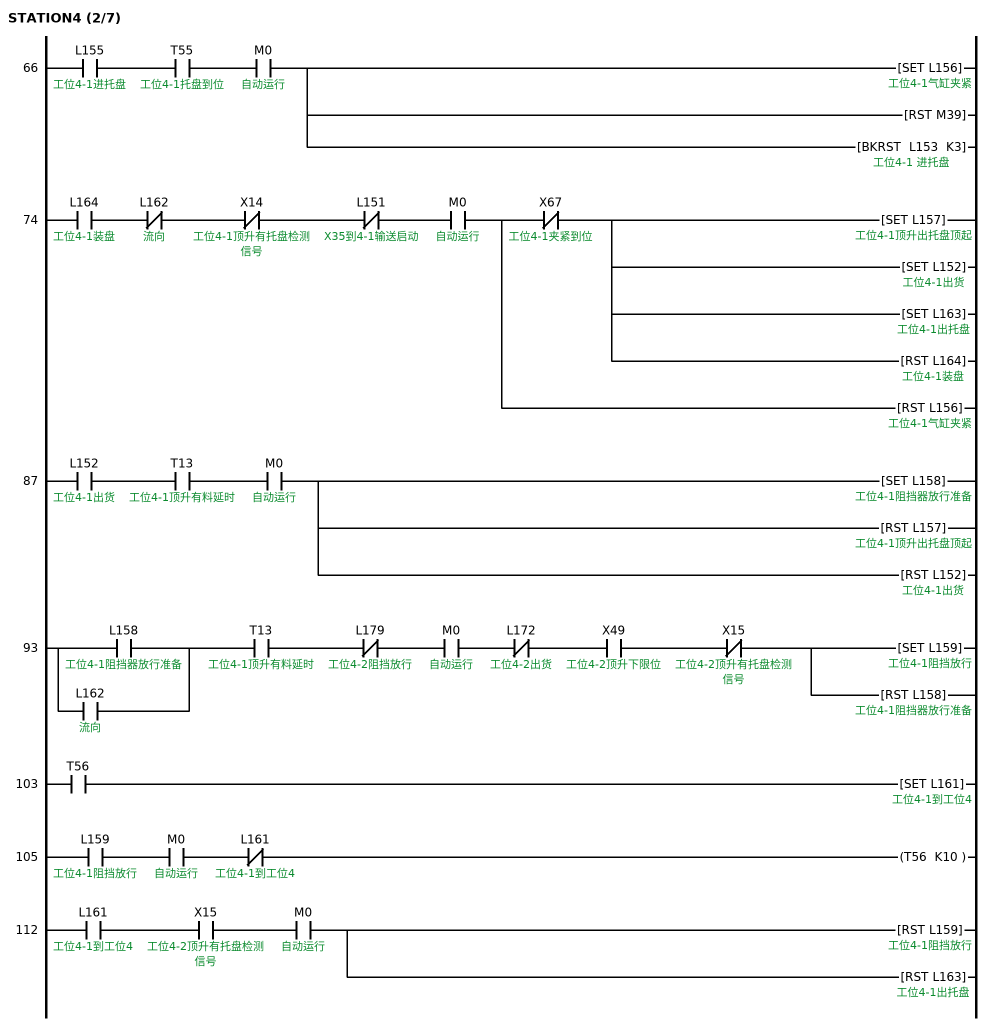
[picture p48: ladder of STATION4, rungs at steps 66 to 112]
66    LD      L155  ; 工位4-1进托盘
      AND     T55  ; 工位4-1托盘到位
      AND     M0  ; 自动运行
      SET     L156  ; 工位4-1气缸夹紧
      RST     M39
      BKRST   L153 K3
74    LD      L164  ; 工位4-1装盘
      ANI     L162  ; 流向
      ANI     X14  ; 工位4-1顶升有托盘检测信号
      ANI     L151  ; X35到4-1输送启动
      AND     M0  ; 自动运行
      MPS
      ANI     X67  ; 工位4-1夹紧到位
      SET     L157  ; 工位4-1顶升出托盘顶起
      SET     L152  ; 工位4-1出货
      SET     L163  ; 工位4-1出托盘
      RST     L164  ; 工位4-1装盘
      MPP
      RST     L156  ; 工位4-1气缸夹紧
87    LD      L152  ; 工位4-1出货
      AND     T13  ; 工位4-1顶升有料延时
      AND     M0  ; 自动运行
      SET     L158  ; 工位4-1阻挡器放行准备
      RST     L157  ; 工位4-1顶升出托盘顶起
      RST     L152  ; 工位4-1出货
93    LD      L158  ; 工位4-1阻挡器放行准备
      OR      L162  ; 流向
      AND     T13  ; 工位4-1顶升有料延时
      ANI     L179  ; 工位4-2阻挡放行
      AND     M0  ; 自动运行
      ANI     L172  ; 工位4-2出货
      AND     X49  ; 工位4-2顶升下限位
      ANI     X15  ; 工位4-2顶升有托盘检测信号
      SET     L159  ; 工位4-1阻挡放行
      RST     L158  ; 工位4-1阻挡器放行准备
103   LD      T56
      SET     L161  ; 工位4-1到工位4
105   LD      L159  ; 工位4-1阻挡放行
      AND     M0  ; 自动运行
      ANI     L161  ; 工位4-1到工位4
      OUT     T56 K10
112   LD      L161  ; 工位4-1到工位4
      AND     X15  ; 工位4-2顶升有托盘检测信号
      AND     M0  ; 自动运行
      RST     L159  ; 工位4-1阻挡放行
      RST     L163  ; 工位4-1出托盘
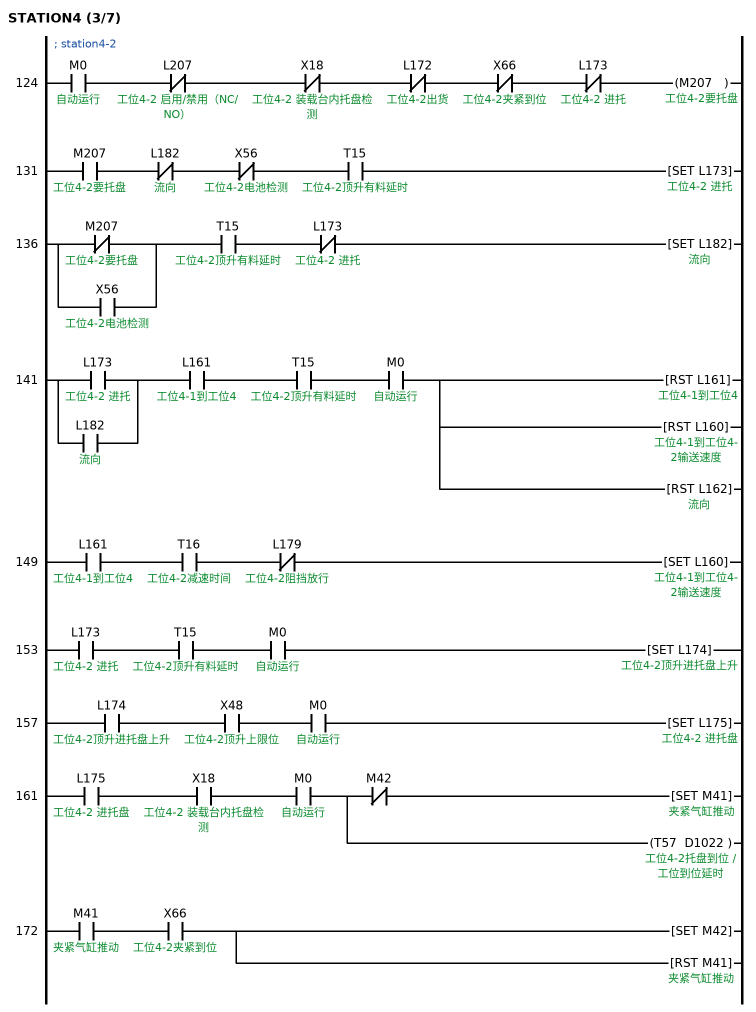
; station4-2
124   LD      M0  ; 自动运行
      ANI     L207  ; 工位4-2 启用/禁用（NC/NO）
      ANI     X18  ; 工位4-2 装载台内托盘检测
      ANI     L172  ; 工位4-2出货
      ANI     X66  ; 工位4-2夹紧到位
      ANI     L173  ; 工位4-2 进托
      OUT     M207  ; 工位4-2要托盘
131   LD      M207  ; 工位4-2要托盘
      ANI     L182  ; 流向
      ANI     X56  ; 工位4-2电池检测
      AND     T15  ; 工位4-2顶升有料延时
      SET     L173  ; 工位4-2 进托
136   LDI     M207  ; 工位4-2要托盘
      OR      X56  ; 工位4-2电池检测
      AND     T15  ; 工位4-2顶升有料延时
      ANI     L173  ; 工位4-2 进托
      SET     L182  ; 流向
141   LD      L173  ; 工位4-2 进托
      OR      L182  ; 流向
      AND     L161  ; 工位4-1到工位4
      AND     T15  ; 工位4-2顶升有料延时
      AND     M0  ; 自动运行
      RST     L161  ; 工位4-1到工位4
      RST     L160  ; 工位4-1到工位4-2输送速度
      RST     L162  ; 流向
149   LD      L161  ; 工位4-1到工位4
      AND     T16  ; 工位4-2减速时间
      ANI     L179  ; 工位4-2阻挡放行
      SET     L160  ; 工位4-1到工位4-2输送速度
153   LD      L173  ; 工位4-2 进托
      AND     T15  ; 工位4-2顶升有料延时
      AND     M0  ; 自动运行
      SET     L174  ; 工位4-2顶升进托盘上升
157   LD      L174  ; 工位4-2顶升进托盘上升
      AND     X48  ; 工位4-2顶升上限位
      AND     M0  ; 自动运行
      SET     L175  ; 工位4-2 进托盘
161   LD      L175  ; 工位4-2 进托盘
      AND     X18  ; 工位4-2 装载台内托盘检测
      AND     M0  ; 自动运行
      MPS
      ANI     M42
      SET     M41  ; 夹紧气缸推动
      MPP
      OUT     T57 D1022  ; 工位4-2托盘到位 / 工位到位延时
172   LD      M41  ; 夹紧气缸推动
      AND     X66  ; 工位4-2夹紧到位
      SET     M42
      RST     M41  ; 夹紧气缸推动
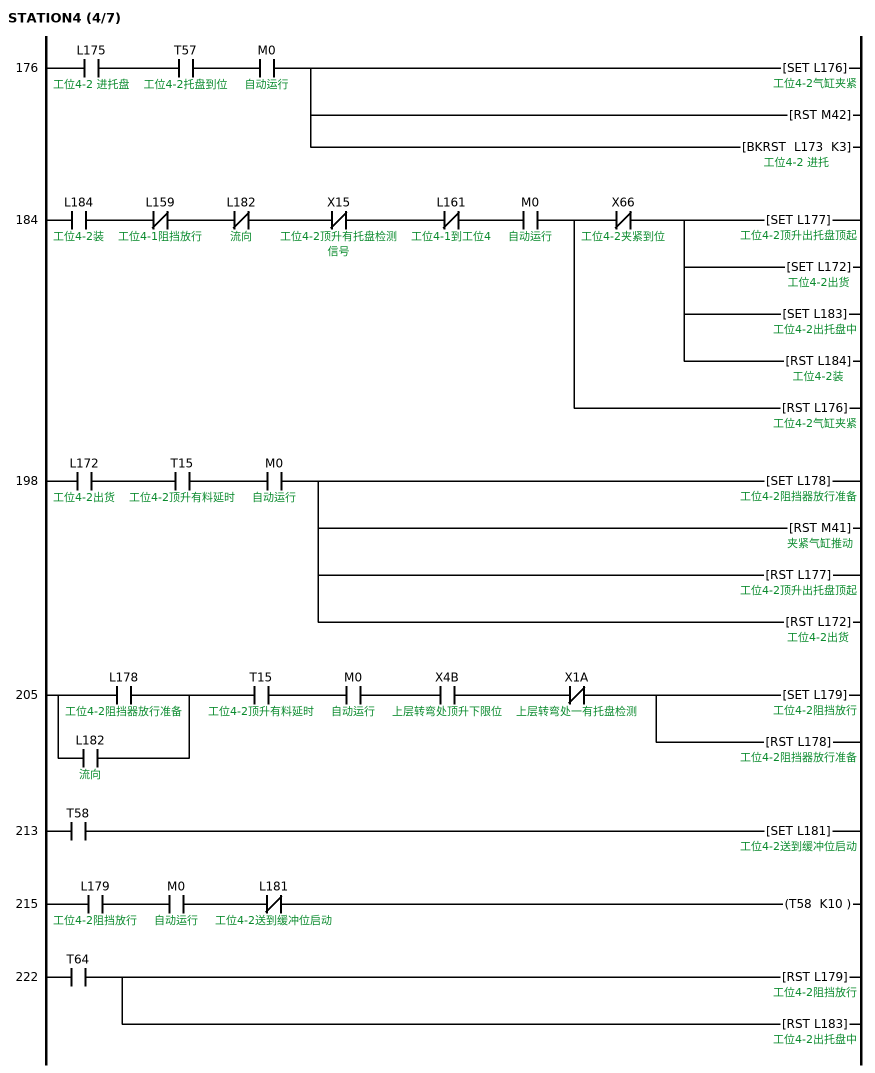
176   LD      L175  ; 工位4-2 进托盘
      AND     T57  ; 工位4-2托盘到位
      AND     M0  ; 自动运行
      SET     L176  ; 工位4-2气缸夹紧
      RST     M42
      BKRST   L173 K3
184   LD      L184  ; 工位4-2装
      ANI     L159  ; 工位4-1阻挡放行
      ANI     L182  ; 流向
      ANI     X15  ; 工位4-2顶升有托盘检测信号
      ANI     L161  ; 工位4-1到工位4
      AND     M0  ; 自动运行
      MPS
      ANI     X66  ; 工位4-2夹紧到位
      SET     L177  ; 工位4-2顶升出托盘顶起
      SET     L172  ; 工位4-2出货
      SET     L183  ; 工位4-2出托盘中
      RST     L184  ; 工位4-2装
      MPP
      RST     L176  ; 工位4-2气缸夹紧
198   LD      L172  ; 工位4-2出货
      AND     T15  ; 工位4-2顶升有料延时
      AND     M0  ; 自动运行
      SET     L178  ; 工位4-2阻挡器放行准备
      RST     M41  ; 夹紧气缸推动
      RST     L177  ; 工位4-2顶升出托盘顶起
      RST     L172  ; 工位4-2出货
205   LD      L178  ; 工位4-2阻挡器放行准备
      OR      L182  ; 流向
      AND     T15  ; 工位4-2顶升有料延时
      AND     M0  ; 自动运行
      AND     X4B  ; 上层转弯处顶升下限位
      ANI     X1A  ; 上层转弯处一有托盘检测
      SET     L179  ; 工位4-2阻挡放行
      RST     L178  ; 工位4-2阻挡器放行准备
213   LD      T58
      SET     L181  ; 工位4-2送到缓冲位启动
215   LD      L179  ; 工位4-2阻挡放行
      AND     M0  ; 自动运行
      ANI     L181  ; 工位4-2送到缓冲位启动
      OUT     T58 K10
222   LD      T64
      RST     L179  ; 工位4-2阻挡放行
      RST     L183  ; 工位4-2出托盘中
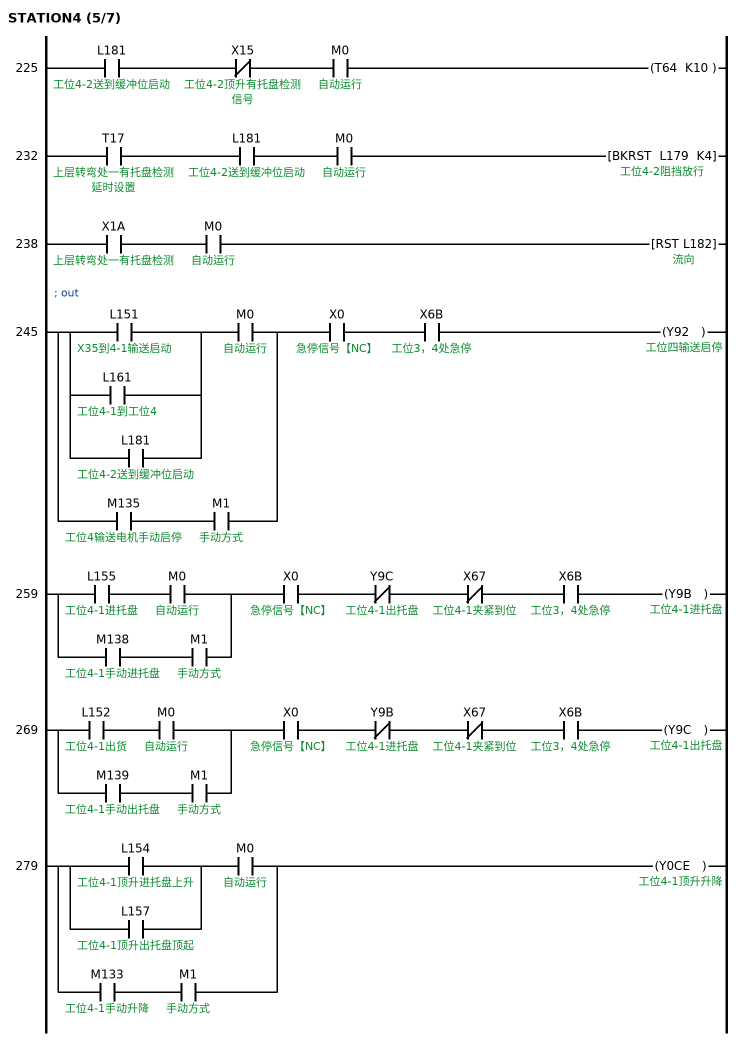
225   LD      L181  ; 工位4-2送到缓冲位启动
      ANI     X15  ; 工位4-2顶升有托盘检测信号
      AND     M0  ; 自动运行
      OUT     T64 K10
232   LD      T17  ; 上层转弯处一有托盘检测延时设置
      AND     L181  ; 工位4-2送到缓冲位启动
      AND     M0  ; 自动运行
      BKRST   L179 K4
238   LD      X1A  ; 上层转弯处一有托盘检测
      AND     M0  ; 自动运行
      RST     L182  ; 流向
; out
245   LD      L151  ; X35到4-1输送启动
      OR      L161  ; 工位4-1到工位4
      OR      L181  ; 工位4-2送到缓冲位启动
      AND     M0  ; 自动运行
      LD      M135  ; 工位4输送电机手动启停
      AND     M1  ; 手动方式
      ORB
      AND     X0  ; 急停信号【NC】
      AND     X6B  ; 工位3，4处急停
      OUT     Y92  ; 工位四输送启停
        [note] 4-1
259   LD      L155  ; 工位4-1进托盘
      AND     M0  ; 自动运行
      LD      M138  ; 工位4-1手动进托盘
      AND     M1  ; 手动方式
      ORB
      AND     X0  ; 急停信号【NC】
      ANI     Y9C  ; 工位4-1出托盘
      ANI     X67  ; 工位4-1夹紧到位
      AND     X6B  ; 工位3，4处急停
      OUT     Y9B  ; 工位4-1进托盘
269   LD      L152  ; 工位4-1出货
      AND     M0  ; 自动运行
      LD      M139  ; 工位4-1手动出托盘
      AND     M1  ; 手动方式
      ORB
      AND     X0  ; 急停信号【NC】
      ANI     Y9B  ; 工位4-1进托盘
      ANI     X67  ; 工位4-1夹紧到位
      AND     X6B  ; 工位3，4处急停
      OUT     Y9C  ; 工位4-1出托盘
279   LD      L154  ; 工位4-1顶升进托盘上升
      OR      L157  ; 工位4-1顶升出托盘顶起
      AND     M0  ; 自动运行
      LD      M133  ; 工位4-1手动升降
      AND     M1  ; 手动方式
      ORB
      OUT     Y0CE  ; 工位4-1顶升升降
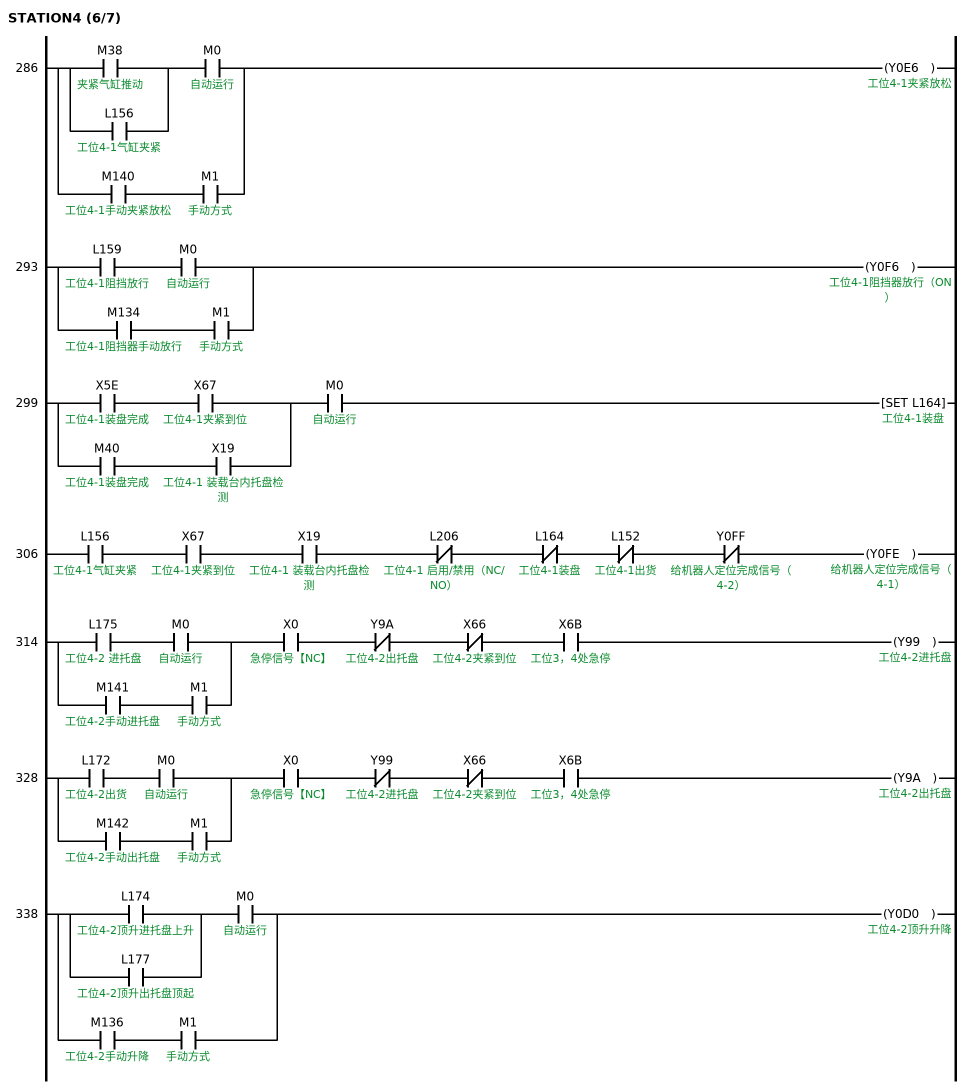
286   LD      M38  ; 夹紧气缸推动
      OR      L156  ; 工位4-1气缸夹紧
      AND     M0  ; 自动运行
      LD      M140  ; 工位4-1手动夹紧放松
      AND     M1  ; 手动方式
      ORB
      OUT     Y0E6  ; 工位4-1夹紧放松
293   LD      L159  ; 工位4-1阻挡放行
      AND     M0  ; 自动运行
      LD      M134  ; 工位4-1阻挡器手动放行
      AND     M1  ; 手动方式
      ORB
      OUT     Y0F6  ; 工位4-1阻挡器放行（ON）
299   LD      X5E  ; 工位4-1装盘完成
      AND     X67  ; 工位4-1夹紧到位
      LD      M40  ; 工位4-1装盘完成
      AND     X19  ; 工位4-1 装载台内托盘检测
      ORB
      AND     M0  ; 自动运行
      SET     L164  ; 工位4-1装盘
306   LD      L156  ; 工位4-1气缸夹紧
      AND     X67  ; 工位4-1夹紧到位
      AND     X19  ; 工位4-1 装载台内托盘检测
      ANI     L206  ; 工位4-1 启用/禁用（NC/NO）
      ANI     L164  ; 工位4-1装盘
      ANI     L152  ; 工位4-1出货
      ANI     Y0FF  ; 给机器人定位完成信号（4-2）
      OUT     Y0FE  ; 给机器人定位完成信号（4-1）
314   LD      L175  ; 工位4-2 进托盘
      AND     M0  ; 自动运行
      LD      M141  ; 工位4-2手动进托盘
      AND     M1  ; 手动方式
      ORB
      AND     X0  ; 急停信号【NC】
      ANI     Y9A  ; 工位4-2出托盘
      ANI     X66  ; 工位4-2夹紧到位
      AND     X6B  ; 工位3，4处急停
      OUT     Y99  ; 工位4-2进托盘
        [note] 4-2
328   LD      L172  ; 工位4-2出货
      AND     M0  ; 自动运行
      LD      M142  ; 工位4-2手动出托盘
      AND     M1  ; 手动方式
      ORB
      AND     X0  ; 急停信号【NC】
      ANI     Y99  ; 工位4-2进托盘
      ANI     X66  ; 工位4-2夹紧到位
      AND     X6B  ; 工位3，4处急停
      OUT     Y9A  ; 工位4-2出托盘
338   LD      L174  ; 工位4-2顶升进托盘上升
      OR      L177  ; 工位4-2顶升出托盘顶起
      AND     M0  ; 自动运行
      LD      M136  ; 工位4-2手动升降
      AND     M1  ; 手动方式
      ORB
      OUT     Y0D0  ; 工位4-2顶升升降
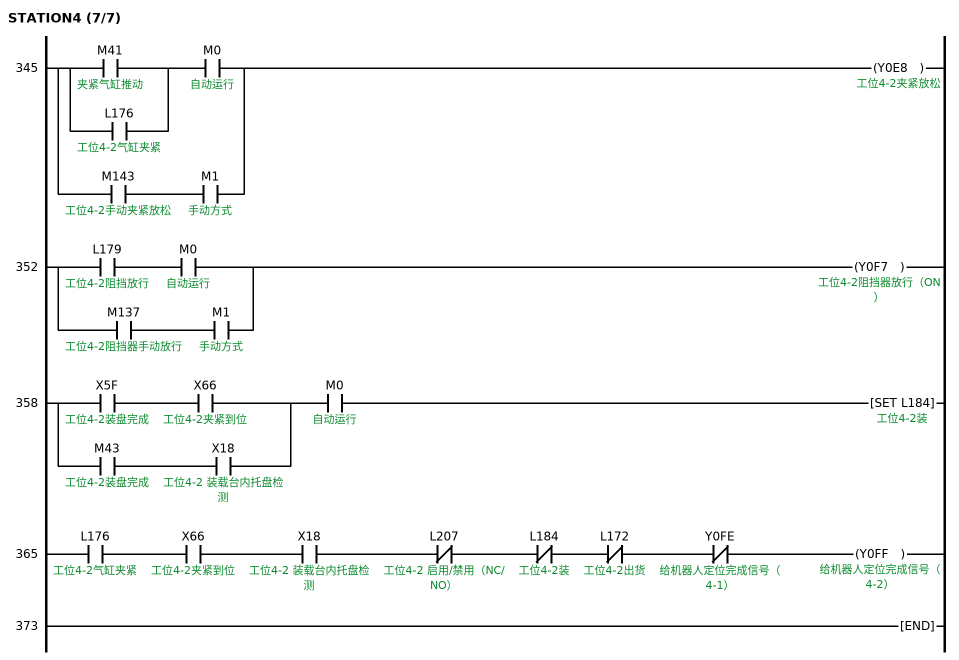
345   LD      M41  ; 夹紧气缸推动
      OR      L176  ; 工位4-2气缸夹紧
      AND     M0  ; 自动运行
      LD      M143  ; 工位4-2手动夹紧放松
      AND     M1  ; 手动方式
      ORB
      OUT     Y0E8  ; 工位4-2夹紧放松
352   LD      L179  ; 工位4-2阻挡放行
      AND     M0  ; 自动运行
      LD      M137  ; 工位4-2阻挡器手动放行
      AND     M1  ; 手动方式
      ORB
      OUT     Y0F7  ; 工位4-2阻挡器放行（ON）
358   LD      X5F  ; 工位4-2装盘完成
      AND     X66  ; 工位4-2夹紧到位
      LD      M43  ; 工位4-2装盘完成
      AND     X18  ; 工位4-2 装载台内托盘检测
      ORB
      AND     M0  ; 自动运行
      SET     L184  ; 工位4-2装
365   LD      L176  ; 工位4-2气缸夹紧
      AND     X66  ; 工位4-2夹紧到位
      AND     X18  ; 工位4-2 装载台内托盘检测
      ANI     L207  ; 工位4-2 启用/禁用（NC/NO）
      ANI     L184  ; 工位4-2装
      ANI     L172  ; 工位4-2出货
      ANI     Y0FE  ; 给机器人定位完成信号（4-1）
      OUT     Y0FF  ; 给机器人定位完成信号（4-2）
373   END
END_PROGRAM

PROGRAM DW-LINE
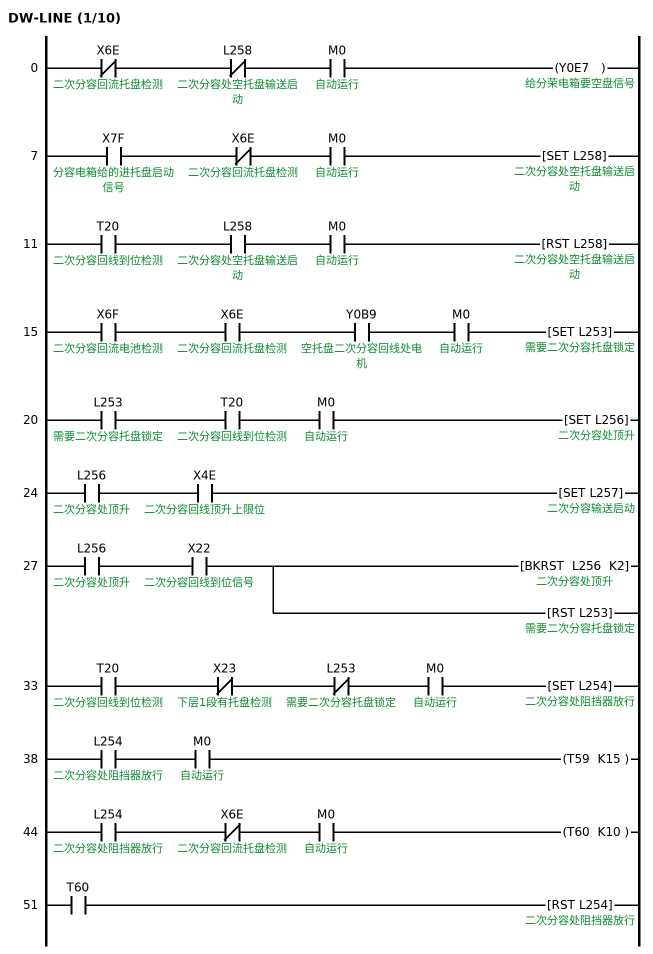
0     LDI     X6E  ; 二次分容回流托盘检测
      ANI     L258  ; 二次分容处空托盘输送启动
      AND     M0  ; 自动运行
      OUT     Y0E7  ; 给分荣电箱要空盘信号
        [note] 1
7     LD      X7F  ; 分容电箱给的进托盘启动信号
      ANI     X6E  ; 二次分容回流托盘检测
      AND     M0  ; 自动运行
      SET     L258  ; 二次分容处空托盘输送启动
11    LD      T20  ; 二次分容回线到位检测
      AND     L258  ; 二次分容处空托盘输送启动
      AND     M0  ; 自动运行
      RST     L258  ; 二次分容处空托盘输送启动
15    LD      X6F  ; 二次分容回流电池检测
      AND     X6E  ; 二次分容回流托盘检测
      AND     Y0B9  ; 空托盘二次分容回线处电机
      AND     M0  ; 自动运行
      SET     L253  ; 需要二次分容托盘锁定
20    LD      L253  ; 需要二次分容托盘锁定
      AND     T20  ; 二次分容回线到位检测
      AND     M0  ; 自动运行
      SET     L256  ; 二次分容处顶升
24    LD      L256  ; 二次分容处顶升
      AND     X4E  ; 二次分容回线顶升上限位
      SET     L257  ; 二次分容输送启动
27    LD      L256  ; 二次分容处顶升
      AND     X22  ; 二次分容回线到位信号
      BKRST   L256 K2
      RST     L253  ; 需要二次分容托盘锁定
33    LD      T20  ; 二次分容回线到位检测
      ANI     X23  ; 下层1段有托盘检测
      ANI     L253  ; 需要二次分容托盘锁定
      AND     M0  ; 自动运行
      SET     L254  ; 二次分容处阻挡器放行
38    LD      L254  ; 二次分容处阻挡器放行
      AND     M0  ; 自动运行
      OUT     T59 K15
44    LD      L254  ; 二次分容处阻挡器放行
      ANI     X6E  ; 二次分容回流托盘检测
      AND     M0  ; 自动运行
      OUT     T60 K10
51    LD      T60
      RST     L254  ; 二次分容处阻挡器放行
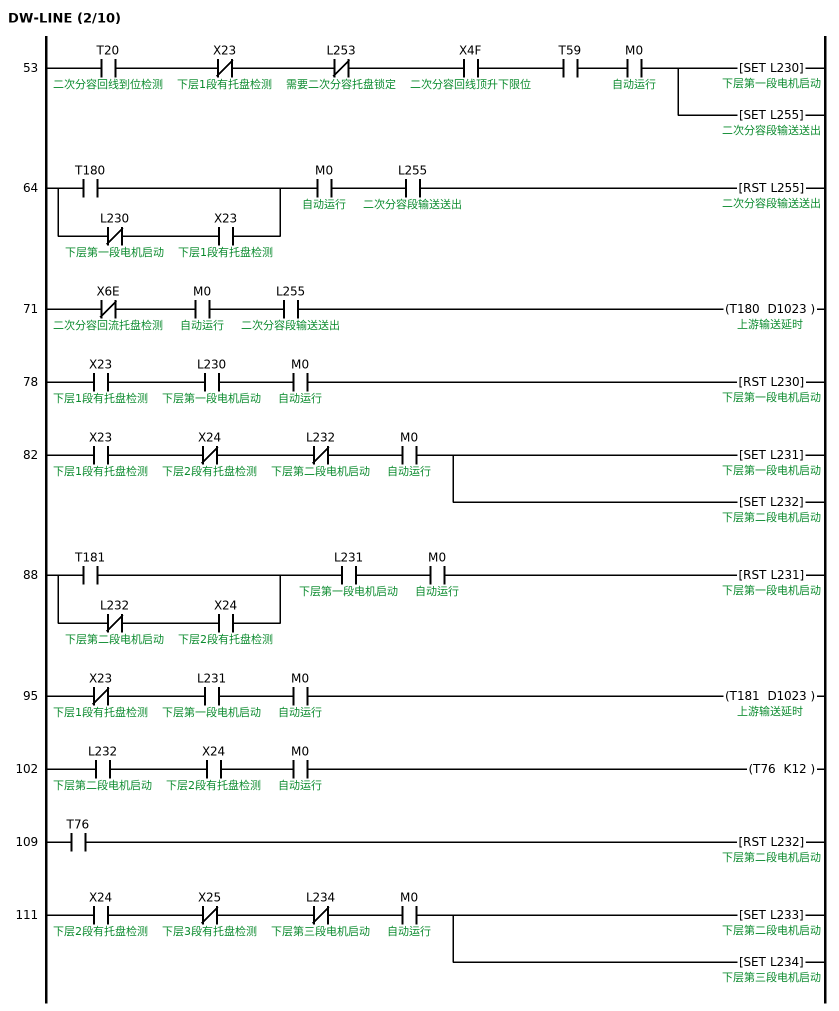
53    LD      T20  ; 二次分容回线到位检测
      ANI     X23  ; 下层1段有托盘检测
      ANI     L253  ; 需要二次分容托盘锁定
      AND     X4F  ; 二次分容回线顶升下限位
      AND     T59
      AND     M0  ; 自动运行
      SET     L230  ; 下层第一段电机启动
        [note] 1
      SET     L255  ; 二次分容段输送送出
64    LD      T180
      LDI     L230  ; 下层第一段电机启动
      AND     X23  ; 下层1段有托盘检测
      ORB
      AND     M0  ; 自动运行
      AND     L255  ; 二次分容段输送送出
      RST     L255  ; 二次分容段输送送出
71    LDI     X6E  ; 二次分容回流托盘检测
      AND     M0  ; 自动运行
      AND     L255  ; 二次分容段输送送出
      OUT     T180 D1023  ; 上游输送延时
78    LD      X23  ; 下层1段有托盘检测
      AND     L230  ; 下层第一段电机启动
      AND     M0  ; 自动运行
      RST     L230  ; 下层第一段电机启动
82    LD      X23  ; 下层1段有托盘检测
      ANI     X24  ; 下层2段有托盘检测
      ANI     L232  ; 下层第二段电机启动
      AND     M0  ; 自动运行
      SET     L231  ; 下层第一段电机启动
      SET     L232  ; 下层第二段电机启动
88    LD      T181
      LDI     L232  ; 下层第二段电机启动
      AND     X24  ; 下层2段有托盘检测
      ORB
      AND     L231  ; 下层第一段电机启动
      AND     M0  ; 自动运行
      RST     L231  ; 下层第一段电机启动
95    LDI     X23  ; 下层1段有托盘检测
      AND     L231  ; 下层第一段电机启动
      AND     M0  ; 自动运行
      OUT     T181 D1023  ; 上游输送延时
102   LD      L232  ; 下层第二段电机启动
      AND     X24  ; 下层2段有托盘检测
      AND     M0  ; 自动运行
      OUT     T76 K12
109   LD      T76
      RST     L232  ; 下层第二段电机启动
111   LD      X24  ; 下层2段有托盘检测
      ANI     X25  ; 下层3段有托盘检测
      ANI     L234  ; 下层第三段电机启动
      AND     M0  ; 自动运行
      SET     L233  ; 下层第二段电机启动
      SET     L234  ; 下层第三段电机启动
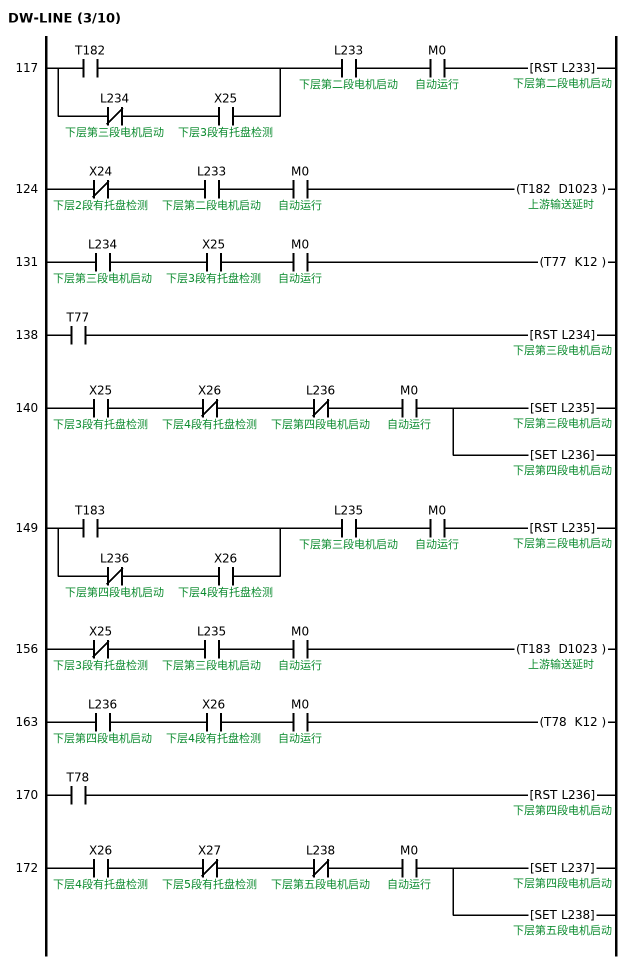
117   LD      T182
      LDI     L234  ; 下层第三段电机启动
      AND     X25  ; 下层3段有托盘检测
      ORB
      AND     L233  ; 下层第二段电机启动
      AND     M0  ; 自动运行
      RST     L233  ; 下层第二段电机启动
124   LDI     X24  ; 下层2段有托盘检测
      AND     L233  ; 下层第二段电机启动
      AND     M0  ; 自动运行
      OUT     T182 D1023  ; 上游输送延时
131   LD      L234  ; 下层第三段电机启动
      AND     X25  ; 下层3段有托盘检测
      AND     M0  ; 自动运行
      OUT     T77 K12
138   LD      T77
      RST     L234  ; 下层第三段电机启动
140   LD      X25  ; 下层3段有托盘检测
      ANI     X26  ; 下层4段有托盘检测
      ANI     L236  ; 下层第四段电机启动
      AND     M0  ; 自动运行
      SET     L235  ; 下层第三段电机启动
        [note] 4
      SET     L236  ; 下层第四段电机启动
149   LD      T183
      LDI     L236  ; 下层第四段电机启动
      AND     X26  ; 下层4段有托盘检测
      ORB
      AND     L235  ; 下层第三段电机启动
      AND     M0  ; 自动运行
      RST     L235  ; 下层第三段电机启动
156   LDI     X25  ; 下层3段有托盘检测
      AND     L235  ; 下层第三段电机启动
      AND     M0  ; 自动运行
      OUT     T183 D1023  ; 上游输送延时
163   LD      L236  ; 下层第四段电机启动
      AND     X26  ; 下层4段有托盘检测
      AND     M0  ; 自动运行
      OUT     T78 K12
170   LD      T78
      RST     L236  ; 下层第四段电机启动
172   LD      X26  ; 下层4段有托盘检测
      ANI     X27  ; 下层5段有托盘检测
      ANI     L238  ; 下层第五段电机启动
      AND     M0  ; 自动运行
      SET     L237  ; 下层第四段电机启动
        [note] 5
      SET     L238  ; 下层第五段电机启动
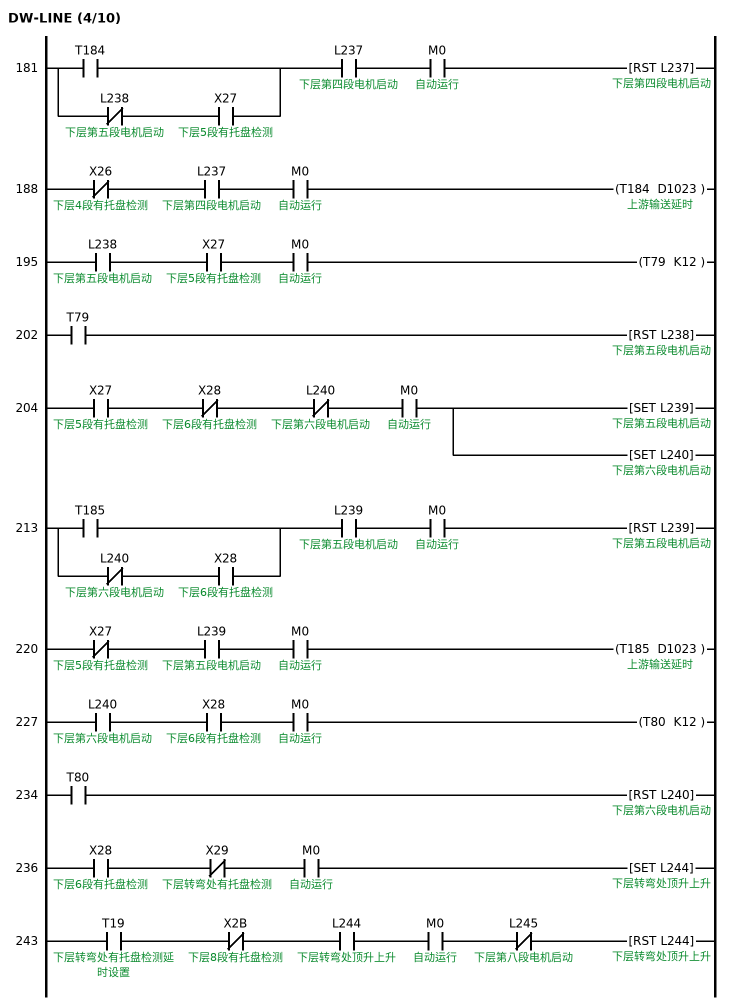
181   LD      T184
      LDI     L238  ; 下层第五段电机启动
      AND     X27  ; 下层5段有托盘检测
      ORB
      AND     L237  ; 下层第四段电机启动
      AND     M0  ; 自动运行
      RST     L237  ; 下层第四段电机启动
188   LDI     X26  ; 下层4段有托盘检测
      AND     L237  ; 下层第四段电机启动
      AND     M0  ; 自动运行
      OUT     T184 D1023  ; 上游输送延时
195   LD      L238  ; 下层第五段电机启动
      AND     X27  ; 下层5段有托盘检测
      AND     M0  ; 自动运行
      OUT     T79 K12
202   LD      T79
      RST     L238  ; 下层第五段电机启动
204   LD      X27  ; 下层5段有托盘检测
      ANI     X28  ; 下层6段有托盘检测
      ANI     L240  ; 下层第六段电机启动
      AND     M0  ; 自动运行
      SET     L239  ; 下层第五段电机启动
        [note] 6
      SET     L240  ; 下层第六段电机启动
213   LD      T185
      LDI     L240  ; 下层第六段电机启动
      AND     X28  ; 下层6段有托盘检测
      ORB
      AND     L239  ; 下层第五段电机启动
      AND     M0  ; 自动运行
      RST     L239  ; 下层第五段电机启动
220   LDI     X27  ; 下层5段有托盘检测
      AND     L239  ; 下层第五段电机启动
      AND     M0  ; 自动运行
      OUT     T185 D1023  ; 上游输送延时
227   LD      L240  ; 下层第六段电机启动
      AND     X28  ; 下层6段有托盘检测
      AND     M0  ; 自动运行
      OUT     T80 K12
234   LD      T80
      RST     L240  ; 下层第六段电机启动
236   LD      X28  ; 下层6段有托盘检测
      ANI     X29  ; 下层转弯处有托盘检测
      AND     M0  ; 自动运行
      SET     L244  ; 下层转弯处顶升上升
        [note] 7
243   LD      T19  ; 下层转弯处有托盘检测延时设置
      ANI     X2B  ; 下层8段有托盘检测
      AND     L244  ; 下层转弯处顶升上升
      AND     M0  ; 自动运行
      ANI     L245  ; 下层第八段电机启动
      RST     L244  ; 下层转弯处顶升上升
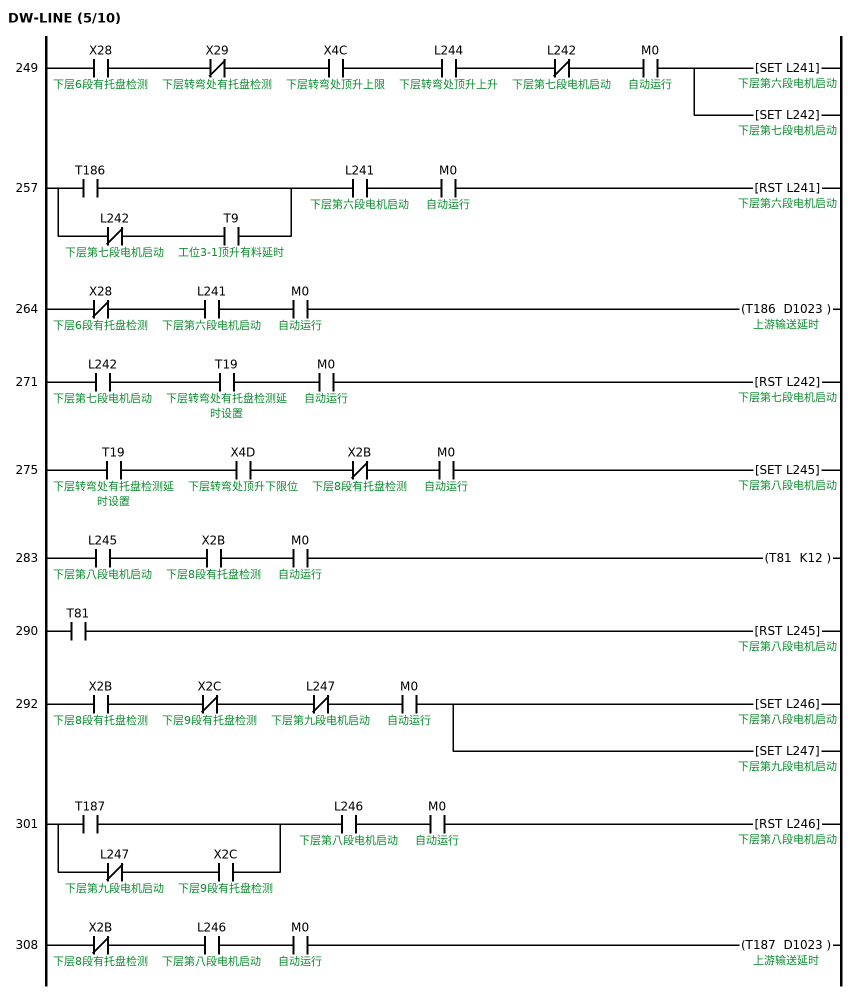
249   LD      X28  ; 下层6段有托盘检测
      ANI     X29  ; 下层转弯处有托盘检测
      AND     X4C  ; 下层转弯处顶升上限
      AND     L244  ; 下层转弯处顶升上升
      ANI     L242  ; 下层第七段电机启动
      AND     M0  ; 自动运行
      SET     L241  ; 下层第六段电机启动
      SET     L242  ; 下层第七段电机启动
257   LD      T186
      LDI     L242  ; 下层第七段电机启动
      AND     T9  ; 工位3-1顶升有料延时
      ORB
      AND     L241  ; 下层第六段电机启动
      AND     M0  ; 自动运行
      RST     L241  ; 下层第六段电机启动
264   LDI     X28  ; 下层6段有托盘检测
      AND     L241  ; 下层第六段电机启动
      AND     M0  ; 自动运行
      OUT     T186 D1023  ; 上游输送延时
271   LD      L242  ; 下层第七段电机启动
      AND     T19  ; 下层转弯处有托盘检测延时设置
      AND     M0  ; 自动运行
      RST     L242  ; 下层第七段电机启动
275   LD      T19  ; 下层转弯处有托盘检测延时设置
      AND     X4D  ; 下层转弯处顶升下限位
      ANI     X2B  ; 下层8段有托盘检测
      AND     M0  ; 自动运行
      SET     L245  ; 下层第八段电机启动
        [note] 8
283   LD      L245  ; 下层第八段电机启动
      AND     X2B  ; 下层8段有托盘检测
      AND     M0  ; 自动运行
      OUT     T81 K12
290   LD      T81
      RST     L245  ; 下层第八段电机启动
292   LD      X2B  ; 下层8段有托盘检测
      ANI     X2C  ; 下层9段有托盘检测
      ANI     L247  ; 下层第九段电机启动
      AND     M0  ; 自动运行
      SET     L246  ; 下层第八段电机启动
        [note] 9
      SET     L247  ; 下层第九段电机启动
301   LD      T187
      LDI     L247  ; 下层第九段电机启动
      AND     X2C  ; 下层9段有托盘检测
      ORB
      AND     L246  ; 下层第八段电机启动
      AND     M0  ; 自动运行
      RST     L246  ; 下层第八段电机启动
308   LDI     X2B  ; 下层8段有托盘检测
      AND     L246  ; 下层第八段电机启动
      AND     M0  ; 自动运行
      OUT     T187 D1023  ; 上游输送延时
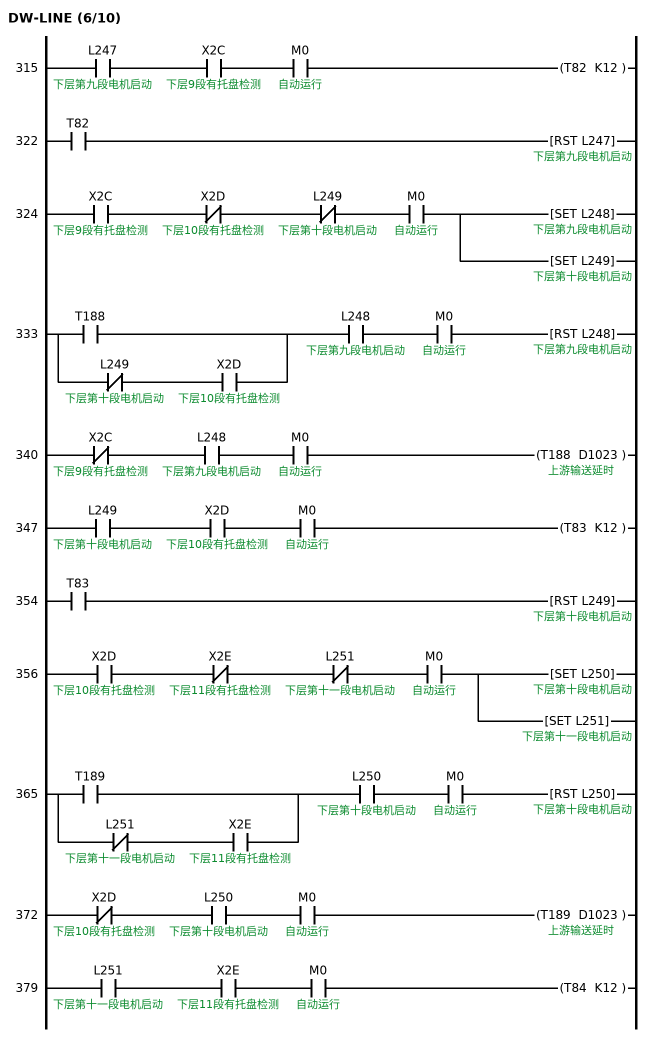
315   LD      L247  ; 下层第九段电机启动
      AND     X2C  ; 下层9段有托盘检测
      AND     M0  ; 自动运行
      OUT     T82 K12
322   LD      T82
      RST     L247  ; 下层第九段电机启动
324   LD      X2C  ; 下层9段有托盘检测
      ANI     X2D  ; 下层10段有托盘检测
      ANI     L249  ; 下层第十段电机启动
      AND     M0  ; 自动运行
      SET     L248  ; 下层第九段电机启动
        [note] 10
      SET     L249  ; 下层第十段电机启动
333   LD      T188
      LDI     L249  ; 下层第十段电机启动
      AND     X2D  ; 下层10段有托盘检测
      ORB
      AND     L248  ; 下层第九段电机启动
      AND     M0  ; 自动运行
      RST     L248  ; 下层第九段电机启动
340   LDI     X2C  ; 下层9段有托盘检测
      AND     L248  ; 下层第九段电机启动
      AND     M0  ; 自动运行
      OUT     T188 D1023  ; 上游输送延时
347   LD      L249  ; 下层第十段电机启动
      AND     X2D  ; 下层10段有托盘检测
      AND     M0  ; 自动运行
      OUT     T83 K12
354   LD      T83
      RST     L249  ; 下层第十段电机启动
356   LD      X2D  ; 下层10段有托盘检测
      ANI     X2E  ; 下层11段有托盘检测
      ANI     L251  ; 下层第十一段电机启动
      AND     M0  ; 自动运行
      SET     L250  ; 下层第十段电机启动
        [note] 10
      SET     L251  ; 下层第十一段电机启动
365   LD      T189
      LDI     L251  ; 下层第十一段电机启动
      AND     X2E  ; 下层11段有托盘检测
      ORB
      AND     L250  ; 下层第十段电机启动
      AND     M0  ; 自动运行
      RST     L250  ; 下层第十段电机启动
372   LDI     X2D  ; 下层10段有托盘检测
      AND     L250  ; 下层第十段电机启动
      AND     M0  ; 自动运行
      OUT     T189 D1023  ; 上游输送延时
379   LD      L251  ; 下层第十一段电机启动
      AND     X2E  ; 下层11段有托盘检测
      AND     M0  ; 自动运行
      OUT     T84 K12
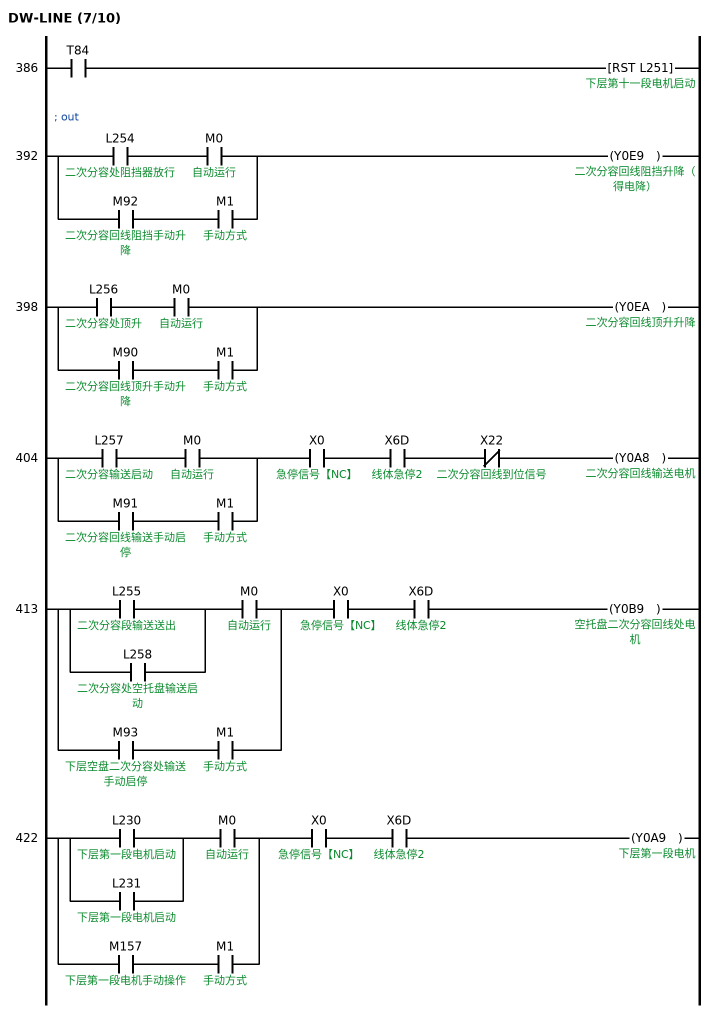
386   LD      T84
      RST     L251  ; 下层第十一段电机启动
; out
392   LD      L254  ; 二次分容处阻挡器放行
      AND     M0  ; 自动运行
      LD      M92  ; 二次分容回线阻挡手动升降
      AND     M1  ; 手动方式
      ORB
      OUT     Y0E9  ; 二次分容回线阻挡升降（得电降）
398   LD      L256  ; 二次分容处顶升
      AND     M0  ; 自动运行
      LD      M90  ; 二次分容回线顶升手动升降
      AND     M1  ; 手动方式
      ORB
      OUT     Y0EA  ; 二次分容回线顶升升降
404   LD      L257  ; 二次分容输送启动
      AND     M0  ; 自动运行
      LD      M91  ; 二次分容回线输送手动启停
      AND     M1  ; 手动方式
      ORB
      AND     X0  ; 急停信号【NC】
      AND     X6D  ; 线体急停2
      ANI     X22  ; 二次分容回线到位信号
      OUT     Y0A8  ; 二次分容回线输送电机
413   LD      L255  ; 二次分容段输送送出
      OR      L258  ; 二次分容处空托盘输送启动
      AND     M0  ; 自动运行
      LD      M93  ; 下层空盘二次分容处输送手动启停
      AND     M1  ; 手动方式
      ORB
      AND     X0  ; 急停信号【NC】
      AND     X6D  ; 线体急停2
      OUT     Y0B9  ; 空托盘二次分容回线处电机
422   LD      L230  ; 下层第一段电机启动
      OR      L231  ; 下层第一段电机启动
      AND     M0  ; 自动运行
      LD      M157  ; 下层第一段电机手动操作
      AND     M1  ; 手动方式
      ORB
      AND     X0  ; 急停信号【NC】
      AND     X6D  ; 线体急停2
      OUT     Y0A9  ; 下层第一段电机
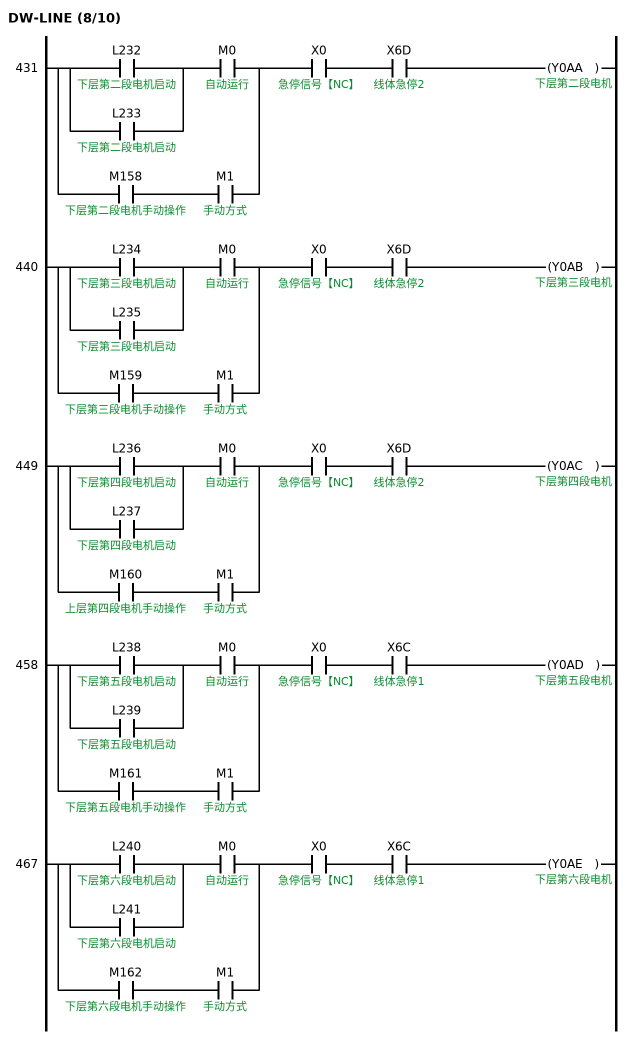
431   LD      L232  ; 下层第二段电机启动
      OR      L233  ; 下层第二段电机启动
      AND     M0  ; 自动运行
      LD      M158  ; 下层第二段电机手动操作
      AND     M1  ; 手动方式
      ORB
      AND     X0  ; 急停信号【NC】
      AND     X6D  ; 线体急停2
      OUT     Y0AA  ; 下层第二段电机
440   LD      L234  ; 下层第三段电机启动
      OR      L235  ; 下层第三段电机启动
      AND     M0  ; 自动运行
      LD      M159  ; 下层第三段电机手动操作
      AND     M1  ; 手动方式
      ORB
      AND     X0  ; 急停信号【NC】
      AND     X6D  ; 线体急停2
      OUT     Y0AB  ; 下层第三段电机
449   LD      L236  ; 下层第四段电机启动
      OR      L237  ; 下层第四段电机启动
      AND     M0  ; 自动运行
      LD      M160  ; 上层第四段电机手动操作
      AND     M1  ; 手动方式
      ORB
      AND     X0  ; 急停信号【NC】
      AND     X6D  ; 线体急停2
      OUT     Y0AC  ; 下层第四段电机
458   LD      L238  ; 下层第五段电机启动
      OR      L239  ; 下层第五段电机启动
      AND     M0  ; 自动运行
      LD      M161  ; 下层第五段电机手动操作
      AND     M1  ; 手动方式
      ORB
      AND     X0  ; 急停信号【NC】
      AND     X6C  ; 线体急停1
      OUT     Y0AD  ; 下层第五段电机
467   LD      L240  ; 下层第六段电机启动
      OR      L241  ; 下层第六段电机启动
      AND     M0  ; 自动运行
      LD      M162  ; 下层第六段电机手动操作
      AND     M1  ; 手动方式
      ORB
      AND     X0  ; 急停信号【NC】
      AND     X6C  ; 线体急停1
      OUT     Y0AE  ; 下层第六段电机
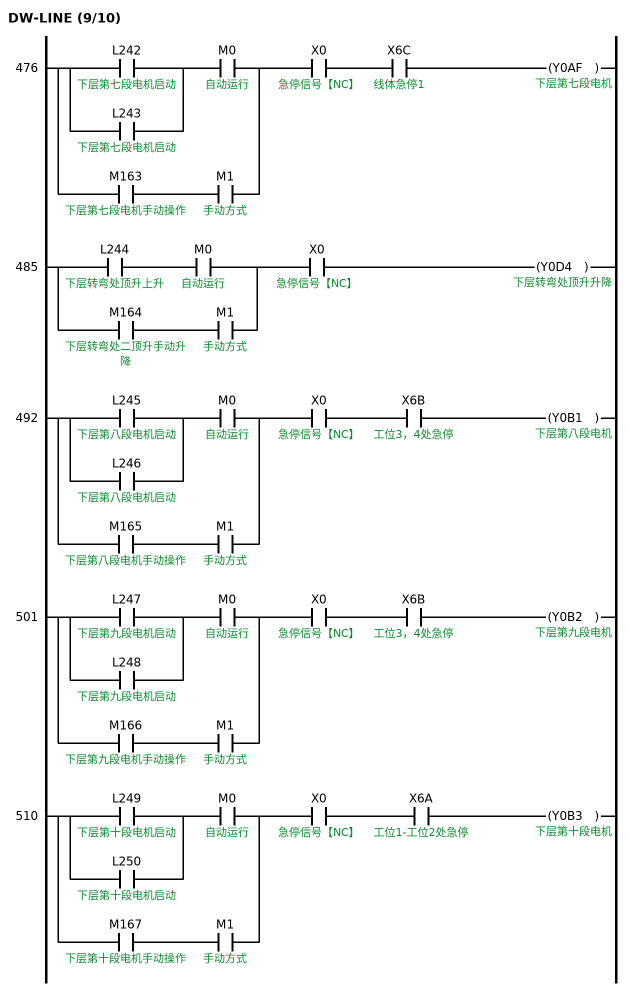
476   LD      L242  ; 下层第七段电机启动
      OR      L243  ; 下层第七段电机启动
      AND     M0  ; 自动运行
      LD      M163  ; 下层第七段电机手动操作
      AND     M1  ; 手动方式
      ORB
      AND     X0  ; 急停信号【NC】
      AND     X6C  ; 线体急停1
      OUT     Y0AF  ; 下层第七段电机
485   LD      L244  ; 下层转弯处顶升上升
      AND     M0  ; 自动运行
      LD      M164  ; 下层转弯处二顶升手动升降
      AND     M1  ; 手动方式
      ORB
      AND     X0  ; 急停信号【NC】
      OUT     Y0D4  ; 下层转弯处顶升升降
492   LD      L245  ; 下层第八段电机启动
      OR      L246  ; 下层第八段电机启动
      AND     M0  ; 自动运行
      LD      M165  ; 下层第八段电机手动操作
      AND     M1  ; 手动方式
      ORB
      AND     X0  ; 急停信号【NC】
      AND     X6B  ; 工位3，4处急停
      OUT     Y0B1  ; 下层第八段电机
501   LD      L247  ; 下层第九段电机启动
      OR      L248  ; 下层第九段电机启动
      AND     M0  ; 自动运行
      LD      M166  ; 下层第九段电机手动操作
      AND     M1  ; 手动方式
      ORB
      AND     X0  ; 急停信号【NC】
      AND     X6B  ; 工位3，4处急停
      OUT     Y0B2  ; 下层第九段电机
510   LD      L249  ; 下层第十段电机启动
      OR      L250  ; 下层第十段电机启动
      AND     M0  ; 自动运行
      LD      M167  ; 下层第十段电机手动操作
      AND     M1  ; 手动方式
      ORB
      AND     X0  ; 急停信号【NC】
      AND     X6A  ; 工位1-工位2处急停
      OUT     Y0B3  ; 下层第十段电机
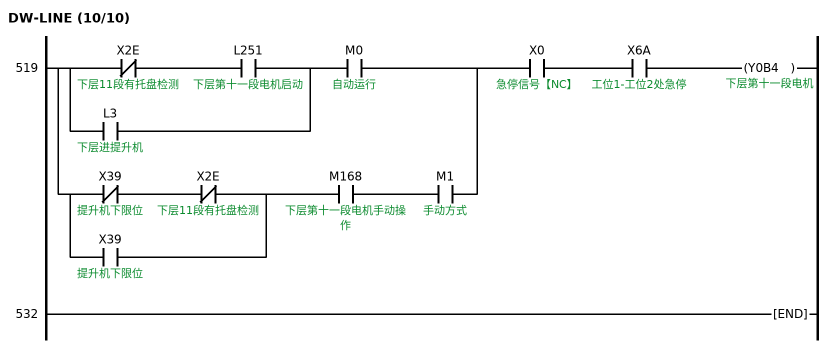
519   LDI     X2E  ; 下层11段有托盘检测
      AND     L251  ; 下层第十一段电机启动
      OR      L3  ; 下层进提升机
      AND     M0  ; 自动运行
      LDI     X39  ; 提升机下限位
      ANI     X2E  ; 下层11段有托盘检测
      OR      X39  ; 提升机下限位
      AND     M168  ; 下层第十一段电机手动操作
      AND     M1  ; 手动方式
      ORB
      AND     X0  ; 急停信号【NC】
      AND     X6A  ; 工位1-工位2处急停
      OUT     Y0B4  ; 下层第十一段电机
532   END
END_PROGRAM

PROGRAM PRODUCT
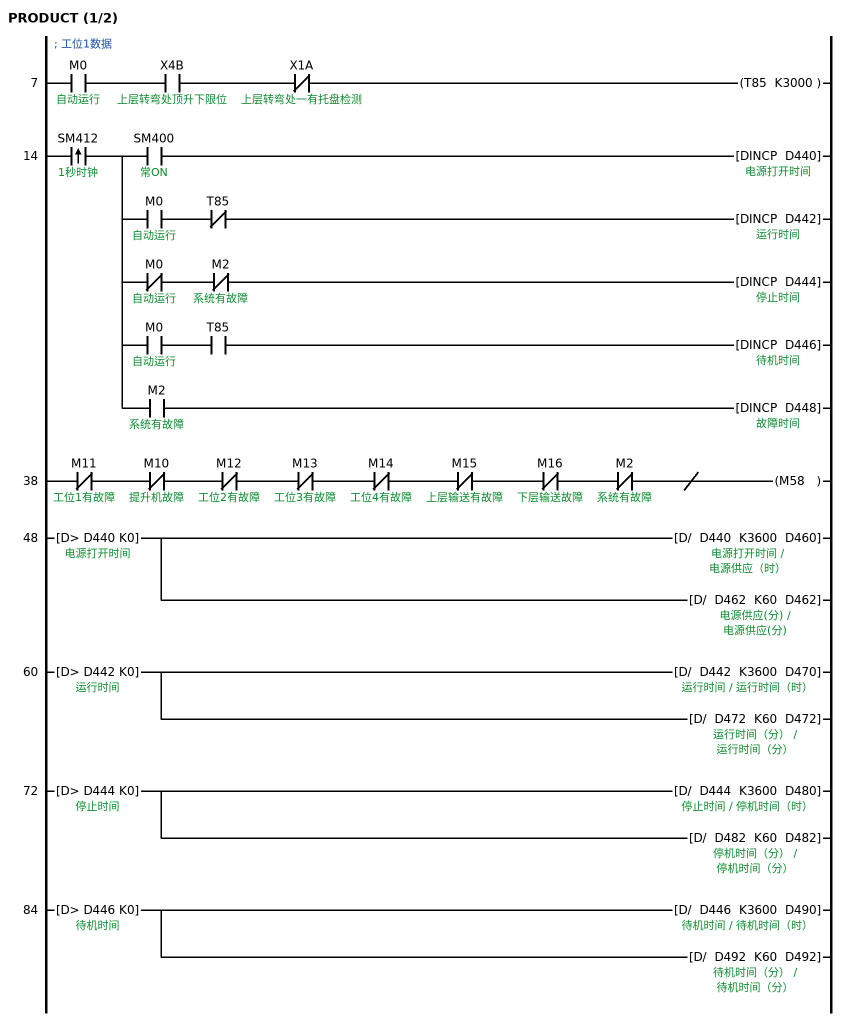
; 工位1数据
7     LD      M0  ; 自动运行
      AND     X4B  ; 上层转弯处顶升下限位
      ANI     X1A  ; 上层转弯处一有托盘检测
      OUT     T85 K3000
14    LDP     SM412  ; 1秒时钟
      MPS
      AND     SM400  ; 常ON
      DINCP   D440  ; 电源打开时间
      MRD
      AND     M0  ; 自动运行
      ANI     T85
      DINCP   D442  ; 运行时间
      MRD
      ANI     M0  ; 自动运行
      ANI     M2  ; 系统有故障
      DINCP   D444  ; 停止时间
      MRD
      AND     M0  ; 自动运行
      AND     T85
      DINCP   D446  ; 待机时间
      MPP
      AND     M2  ; 系统有故障
      DINCP   D448  ; 故障时间
38    LDI     M11  ; 工位1有故障
      ANI     M10  ; 提升机故障
      ANI     M12  ; 工位2有故障
      ANI     M13  ; 工位3有故障
      ANI     M14  ; 工位4有故障
      ANI     M15  ; 上层输送有故障
      ANI     M16  ; 下层输送故障
      ANI     M2  ; 系统有故障
      INV
      OUT     M58
48    LDD>    D440 K0  ; 电源打开时间
      D/      D440 K3600 D460  ; 电源供应（时）
      D/      D462 K60 D462  ; 电源供应(分)
60    LDD>    D442 K0  ; 运行时间
      D/      D442 K3600 D470  ; 运行时间（时）
      D/      D472 K60 D472  ; 运行时间（分）
72    LDD>    D444 K0  ; 停止时间
      D/      D444 K3600 D480  ; 停机时间（时）
      D/      D482 K60 D482  ; 停机时间（分）
84    LDD>    D446 K0  ; 待机时间
      D/      D446 K3600 D490  ; 待机时间（时）
      D/      D492 K60 D492  ; 待机时间（分）
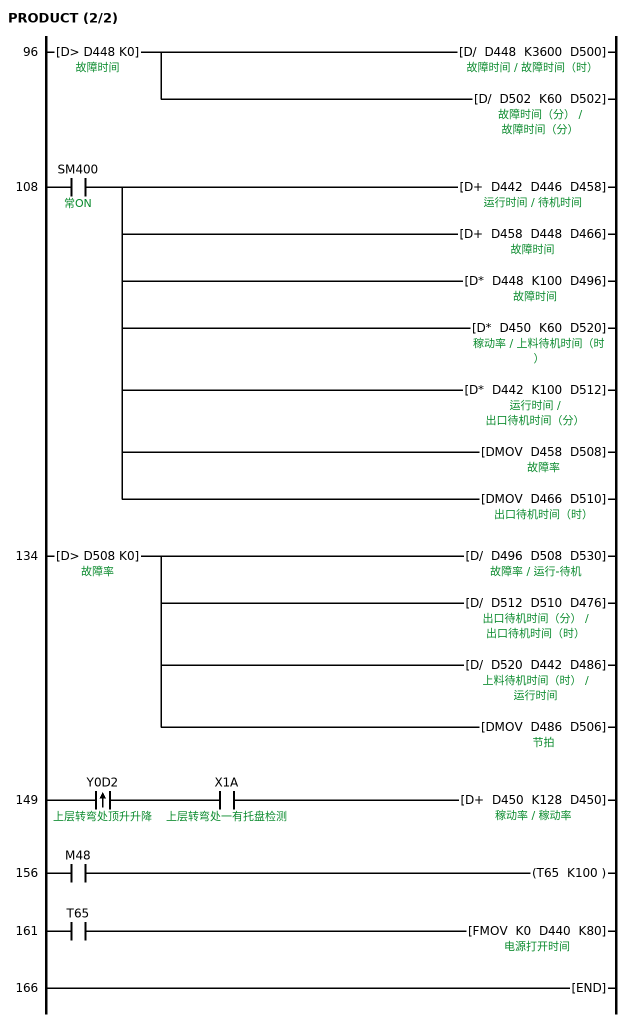
96    LDD>    D448 K0  ; 故障时间
      D/      D448 K3600 D500  ; 故障时间（时）
      D/      D502 K60 D502  ; 故障时间（分）
108   LD      SM400  ; 常ON
      D+      D442 D446 D458
        [note] 秒
      D+      D458 D448 D466
      D*      D448 K100 D496
      D*      D450 K60 D520  ; 稼动率 / 上料待机时间（时）
      D*      D442 K100 D512  ; 出口待机时间（分）
      DMOV    D458 D508  ; 故障率
      DMOV    D466 D510  ; 出口待机时间（时）
134   LDD>    D508 K0  ; 故障率
      D/      D496 D508 D530  ; 运行-待机
      D/      D512 D510 D476
      D/      D520 D442 D486
      DMOV    D486 D506  ; 节拍
149   LDP     Y0D2  ; 上层转弯处顶升升降
      AND     X1A  ; 上层转弯处一有托盘检测
      D+      D450 K128 D450
156   LD      M48
      OUT     T65 K100
161   LD      T65
      FMOV    K0 D440 K80
166   END
END_PROGRAM

PROGRAM MAIN
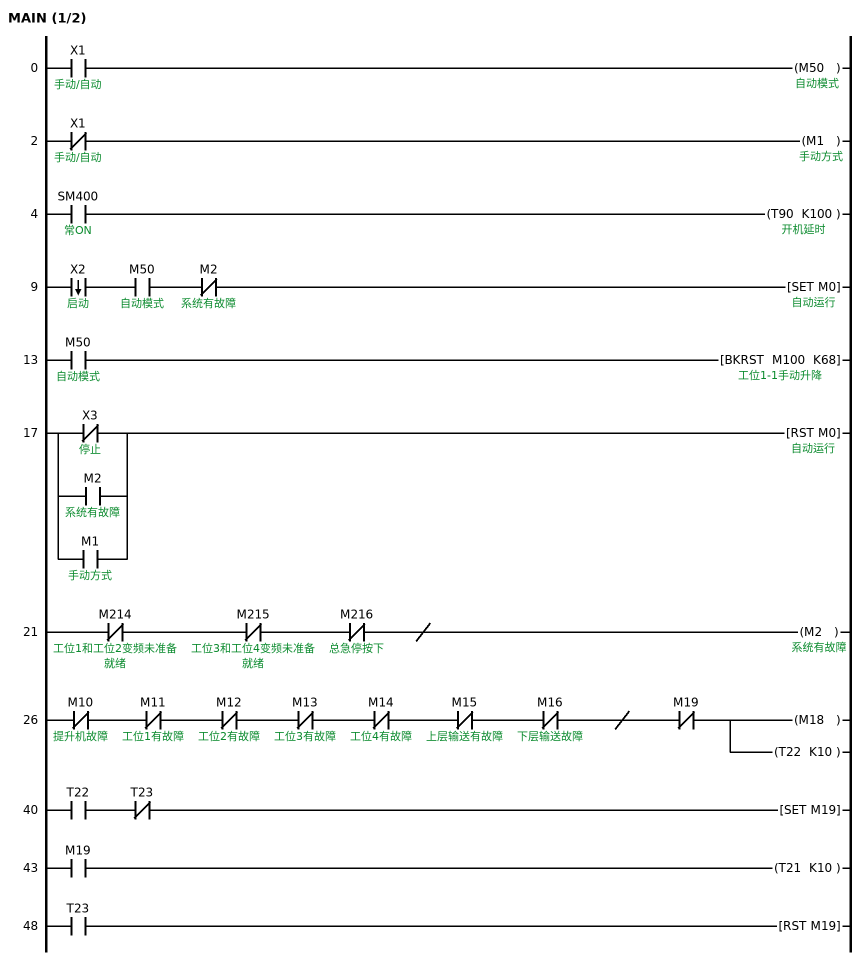
0     LD      X1  ; 手动/自动
      OUT     M50  ; 自动模式
2     LDI     X1  ; 手动/自动
      OUT     M1  ; 手动方式
4     LD      SM400  ; 常ON
      OUT     T90 K100  ; 开机延时
9     LDF     X2  ; 启动
      AND     M50  ; 自动模式
      ANI     M2  ; 系统有故障
      SET     M0  ; 自动运行
13    LD      M50  ; 自动模式
      BKRST   M100 K68  ; 工位1-1手动升降
17    LDI     X3  ; 停止
      OR      M2  ; 系统有故障
      OR      M1  ; 手动方式
      RST     M0  ; 自动运行
21    LDI     M214  ; 工位1和工位2变频未准备就绪
      ANI     M215  ; 工位3和工位4变频未准备就绪
      ANI     M216  ; 总急停按下
      INV
      OUT     M2  ; 系统有故障
26    LDI     M10  ; 提升机故障
      ANI     M11  ; 工位1有故障
      ANI     M12  ; 工位2有故障
      ANI     M13  ; 工位3有故障
      ANI     M14  ; 工位4有故障
      ANI     M15  ; 上层输送有故障
      ANI     M16  ; 下层输送故障
      INV
      ANI     M19
      OUT     M18
      OUT     T22 K10
40    LD      T22
      ANI     T23
      SET     M19
43    LD      M19
      OUT     T21 K10
48    LD      T23
      RST     M19
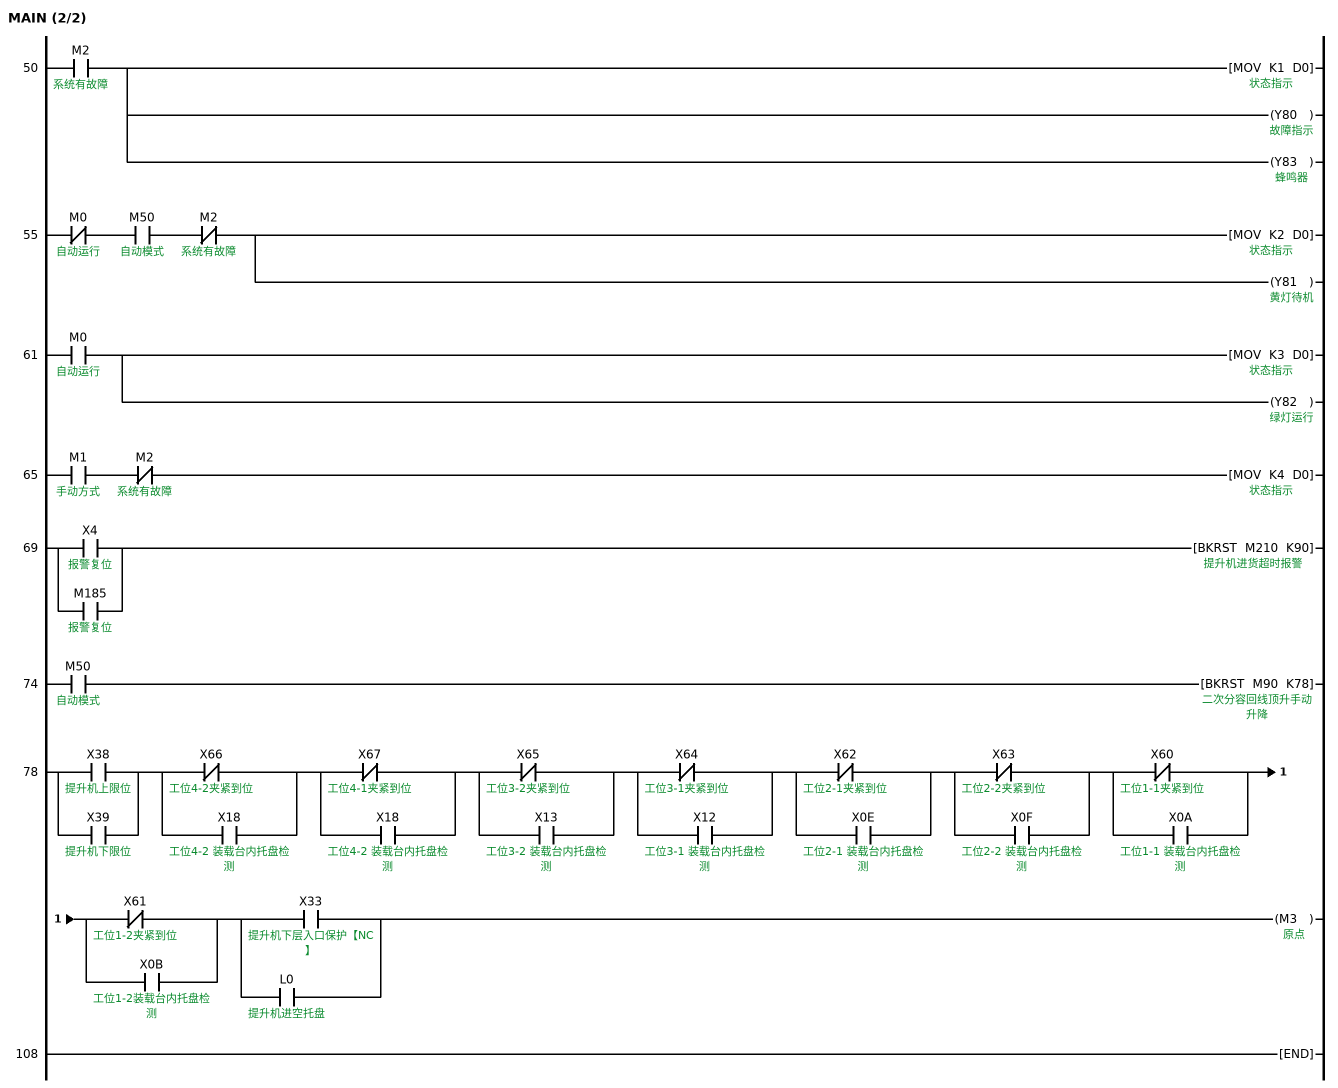
50    LD      M2  ; 系统有故障
      MOV     K1 D0  ; 状态指示
      OUT     Y80  ; 故障指示
      OUT     Y83  ; 蜂鸣器
55    LDI     M0  ; 自动运行
      AND     M50  ; 自动模式
      ANI     M2  ; 系统有故障
      MOV     K2 D0
      OUT     Y81  ; 黄灯待机
61    LD      M0  ; 自动运行
      MOV     K3 D0
      OUT     Y82  ; 绿灯运行
65    LD      M1  ; 手动方式
      ANI     M2  ; 系统有故障
      MOV     K4 D0
69    LD      X4  ; 报警复位
      OR      M185  ; 报警复位
      BKRST   M210 K90  ; 提升机进货超时报警
74    LD      M50  ; 自动模式
      BKRST   M90 K78  ; 二次分容回线顶升手动升降
78    LD      X38  ; 提升机上限位
      OR      X39  ; 提升机下限位
      LDI     X66  ; 工位4-2夹紧到位
      OR      X18  ; 工位4-2 装载台内托盘检测
      ANB
      LDI     X67  ; 工位4-1夹紧到位
      OR      X18  ; 工位4-2 装载台内托盘检测
      ANB
      LDI     X65  ; 工位3-2夹紧到位
      OR      X13  ; 工位3-2 装载台内托盘检测
      ANB
      LDI     X64  ; 工位3-1夹紧到位
      OR      X12  ; 工位3-1 装载台内托盘检测
      ANB
      LDI     X62  ; 工位2-1夹紧到位
      OR      X0E  ; 工位2-1 装载台内托盘检测
      ANB
      LDI     X63  ; 工位2-2夹紧到位
      OR      X0F  ; 工位2-2 装载台内托盘检测
      ANB
      LDI     X60  ; 工位1-1夹紧到位
      OR      X0A  ; 工位1-1 装载台内托盘检测
      ANB
      LDI     X61  ; 工位1-2夹紧到位
      OR      X0B  ; 工位1-2装载台内托盘检测
      ANB
      LD      X33  ; 提升机下层入口保护【NC】
      OR      L0  ; 提升机进空托盘
      ANB
      OUT     M3  ; 原点
108   END
END_PROGRAM

PROGRAM HMITimer
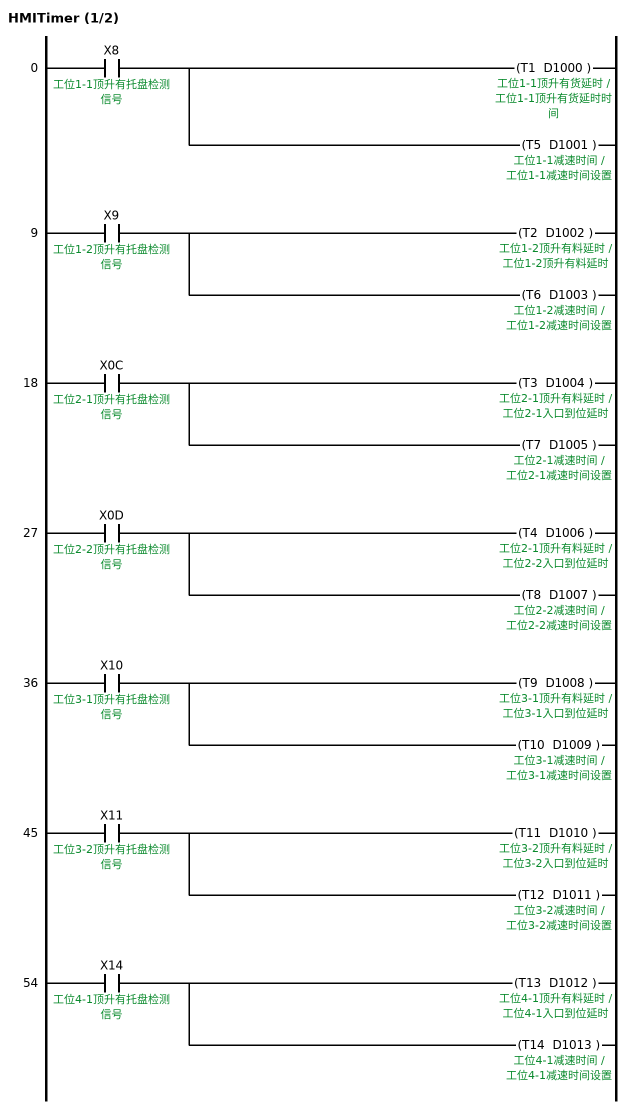
0     LD      X8  ; 工位1-1顶升有托盘检测信号
      OUT     T1 D1000  ; 工位1-1顶升有货延时 / 工位1-1顶升有货延时时间
      OUT     T5 D1001  ; 工位1-1减速时间 / 工位1-1减速时间设置
9     LD      X9  ; 工位1-2顶升有托盘检测信号
      OUT     T2 D1002  ; 工位1-2顶升有料延时 / 工位1-2顶升有料延时
      OUT     T6 D1003  ; 工位1-2减速时间 / 工位1-2减速时间设置
18    LD      X0C  ; 工位2-1顶升有托盘检测信号
      OUT     T3 D1004  ; 工位2-1顶升有料延时 / 工位2-1入口到位延时
      OUT     T7 D1005  ; 工位2-1减速时间 / 工位2-1减速时间设置
27    LD      X0D  ; 工位2-2顶升有托盘检测信号
      OUT     T4 D1006  ; 工位2-1顶升有料延时 / 工位2-2入口到位延时
      OUT     T8 D1007  ; 工位2-2减速时间 / 工位2-2减速时间设置
36    LD      X10  ; 工位3-1顶升有托盘检测信号
      OUT     T9 D1008  ; 工位3-1顶升有料延时 / 工位3-1入口到位延时
      OUT     T10 D1009  ; 工位3-1减速时间 / 工位3-1减速时间设置
45    LD      X11  ; 工位3-2顶升有托盘检测信号
      OUT     T11 D1010  ; 工位3-2顶升有料延时 / 工位3-2入口到位延时
      OUT     T12 D1011  ; 工位3-2减速时间 / 工位3-2减速时间设置
54    LD      X14  ; 工位4-1顶升有托盘检测信号
      OUT     T13 D1012  ; 工位4-1顶升有料延时 / 工位4-1入口到位延时
      OUT     T14 D1013  ; 工位4-1减速时间 / 工位4-1减速时间设置
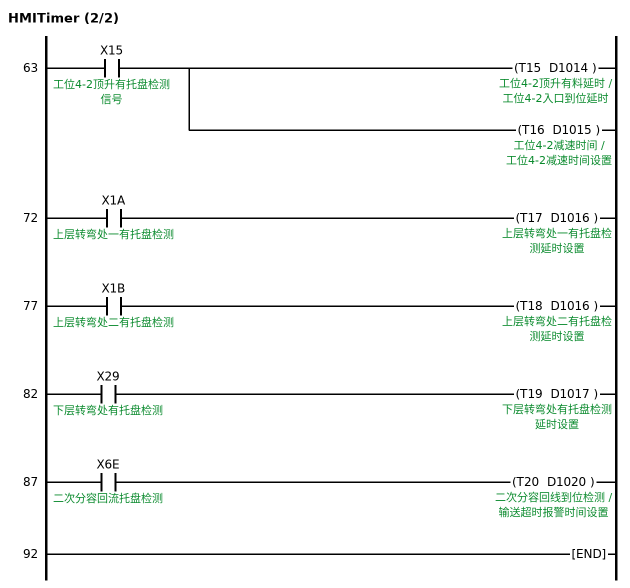
63    LD      X15  ; 工位4-2顶升有托盘检测信号
      OUT     T15 D1014  ; 工位4-2顶升有料延时 / 工位4-2入口到位延时
      OUT     T16 D1015  ; 工位4-2减速时间 / 工位4-2减速时间设置
72    LD      X1A  ; 上层转弯处一有托盘检测
      OUT     T17 D1016  ; 上层转弯处一有托盘检测延时设置
77    LD      X1B  ; 上层转弯处二有托盘检测
      OUT     T18 D1016  ; 上层转弯处二有托盘检测延时设置
82    LD      X29  ; 下层转弯处有托盘检测
      OUT     T19 D1017  ; 下层转弯处有托盘检测延时设置
87    LD      X6E  ; 二次分容回流托盘检测
      OUT     T20 D1020  ; 二次分容回线到位检测 / 输送超时报警时间设置
92    END
END_PROGRAM

PROGRAM TP-LINE
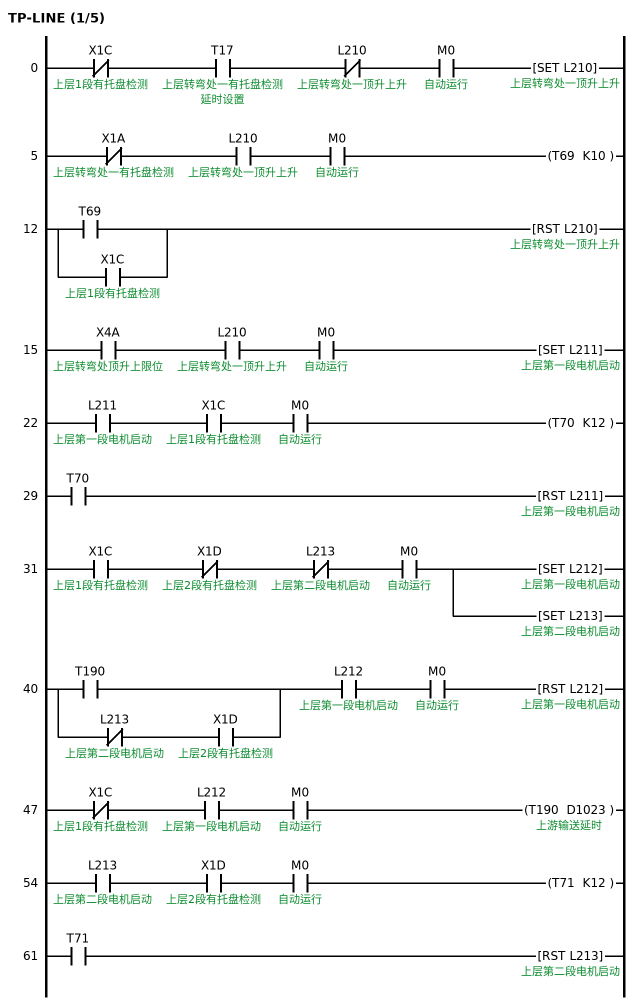
0     LDI     X1C  ; 上层1段有托盘检测
      AND     T17  ; 上层转弯处一有托盘检测延时设置
      ANI     L210  ; 上层转弯处一顶升上升
      AND     M0  ; 自动运行
      SET     L210  ; 上层转弯处一顶升上升
5     LDI     X1A  ; 上层转弯处一有托盘检测
      AND     L210  ; 上层转弯处一顶升上升
      AND     M0  ; 自动运行
      OUT     T69 K10
12    LD      T69
      OR      X1C  ; 上层1段有托盘检测
      RST     L210  ; 上层转弯处一顶升上升
15    LD      X4A  ; 上层转弯处顶升上限位
      AND     L210  ; 上层转弯处一顶升上升
      AND     M0  ; 自动运行
      SET     L211  ; 上层第一段电机启动
        [note] 1
22    LD      L211  ; 上层第一段电机启动
      AND     X1C  ; 上层1段有托盘检测
      AND     M0  ; 自动运行
      OUT     T70 K12
29    LD      T70
      RST     L211  ; 上层第一段电机启动
31    LD      X1C  ; 上层1段有托盘检测
      ANI     X1D  ; 上层2段有托盘检测
      ANI     L213  ; 上层第二段电机启动
      AND     M0  ; 自动运行
      SET     L212  ; 上层第一段电机启动
        [note] 2
      SET     L213  ; 上层第二段电机启动
40    LD      T190
      LDI     L213  ; 上层第二段电机启动
      AND     X1D  ; 上层2段有托盘检测
      ORB
      AND     L212  ; 上层第一段电机启动
      AND     M0  ; 自动运行
      RST     L212  ; 上层第一段电机启动
47    LDI     X1C  ; 上层1段有托盘检测
      AND     L212  ; 上层第一段电机启动
      AND     M0  ; 自动运行
      OUT     T190 D1023  ; 上游输送延时
54    LD      L213  ; 上层第二段电机启动
      AND     X1D  ; 上层2段有托盘检测
      AND     M0  ; 自动运行
      OUT     T71 K12
61    LD      T71
      RST     L213  ; 上层第二段电机启动
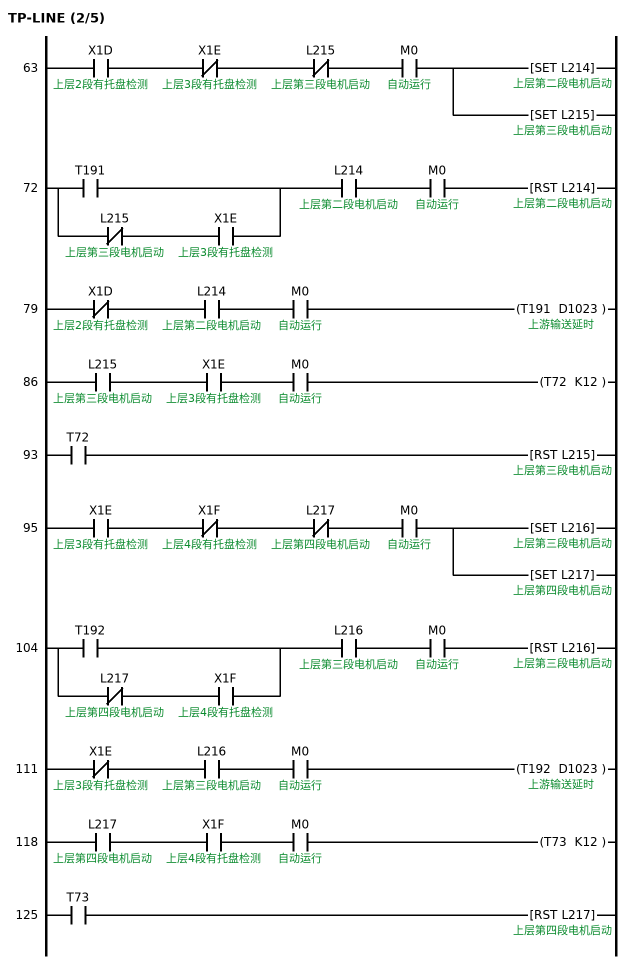
63    LD      X1D  ; 上层2段有托盘检测
      ANI     X1E  ; 上层3段有托盘检测
      ANI     L215  ; 上层第三段电机启动
      AND     M0  ; 自动运行
      SET     L214  ; 上层第二段电机启动
        [note] 3
      SET     L215  ; 上层第三段电机启动
72    LD      T191
      LDI     L215  ; 上层第三段电机启动
      AND     X1E  ; 上层3段有托盘检测
      ORB
      AND     L214  ; 上层第二段电机启动
      AND     M0  ; 自动运行
      RST     L214  ; 上层第二段电机启动
79    LDI     X1D  ; 上层2段有托盘检测
      AND     L214  ; 上层第二段电机启动
      AND     M0  ; 自动运行
      OUT     T191 D1023  ; 上游输送延时
86    LD      L215  ; 上层第三段电机启动
      AND     X1E  ; 上层3段有托盘检测
      AND     M0  ; 自动运行
      OUT     T72 K12
93    LD      T72
      RST     L215  ; 上层第三段电机启动
95    LD      X1E  ; 上层3段有托盘检测
      ANI     X1F  ; 上层4段有托盘检测
      ANI     L217  ; 上层第四段电机启动
      AND     M0  ; 自动运行
      SET     L216  ; 上层第三段电机启动
        [note] 4
      SET     L217  ; 上层第四段电机启动
104   LD      T192
      LDI     L217  ; 上层第四段电机启动
      AND     X1F  ; 上层4段有托盘检测
      ORB
      AND     L216  ; 上层第三段电机启动
      AND     M0  ; 自动运行
      RST     L216  ; 上层第三段电机启动
111   LDI     X1E  ; 上层3段有托盘检测
      AND     L216  ; 上层第三段电机启动
      AND     M0  ; 自动运行
      OUT     T192 D1023  ; 上游输送延时
118   LD      L217  ; 上层第四段电机启动
      AND     X1F  ; 上层4段有托盘检测
      AND     M0  ; 自动运行
      OUT     T73 K12
125   LD      T73
      RST     L217  ; 上层第四段电机启动
